// Motion Pickup n Deposit HW inputs
TYPE ST_HW_InputsMPD :

STRUCT	
	Conv						: ARRAY[1..2] OF ST_HW_InputsMPD_Conv;	
	ManualControl				: ST_HW_InputsManControl;
	DriveInputs					: ST_PDO_DriveIn;	
END_STRUCT
END_TYPE

(* stored: Version 1.1.0.1, ProductVersion 3.1.4024.9
   DUT ST_HW_InputsMPD: Id {581c8f64-b741-43a6-91fa-955c1fed3725} *)
